{attribute addProperty BoxType "EL3773-0000-0016"}
{attribute addProperty Id "U1_STATUSAT %I*U1_STATUS_F9B4A013162"}
{attribute addProperty CRC "598670270"}
{attribute addProperty SizeInBites "16"}
{attribute addProperty SizeInBytes "2"}
TYPE L1_Voltage_Status_23AEFBBE :
STRUCT
	{attribute addProperty Name "U1_STATUS"}
	U1_STATUS AT %I* : U1_STATUS_F9B4A013;
END_STRUCT
END_TYPE

(* stored: Version 1.2.0.0, ProductVersion 3.1.4024.9
   DUT L1_Voltage_Status_23AEFBBE: Id {4a4790e4-c7d1-442b-8045-d2d386db00a6} *)
